FUNCTION WORDS_TO_DWORD
  (* Standard: 61499-1; Description: Copyright (c) 2024 HR Agrartechnik GmbH This program and the accompanying materials are made available under the terms of the Eclipse Public License 2.0 which is available at https://www.eclipse.org/legal/epl-2.0/ SPDX-License-Identifier: EPL-2.0 *)
  (* Version 1.0, 2024-02-22, franz *)
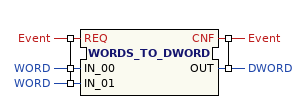
  EVENT_INPUT
    REQ WITH IN_00, IN_01;
  END_EVENT
  EVENT_OUTPUT
    CNF WITH OUT;
  END_EVENT
  VAR_INPUT
    IN_00 : WORD; (* WORD 00 *)
    IN_01 : WORD; (* WORD 01 *)
  END_VAR
  VAR_OUTPUT
    OUT : DWORD; (* DWORD Output *)
  END_VAR
  BODY IN ST:
FUNCTION WORDS_TO_DWORD

VAR_INPUT
	IN_00 : WORD;    // WORD 00
	IN_01 : WORD;    // WORD 01
END_VAR

VAR_OUTPUT
	OUT : DWORD;    // DWORD Output
END_VAR

(* this Function combines the 2 WORDS to a dword *)
OUT := SHL(WORD_TO_DWORD(IN_01), SHIFT_WORD_01)
	OR SHL(WORD_TO_DWORD(IN_00), SHIFT_WORD_00);

END_FUNCTION
  END_BODY
END_FUNCTION
